FUNCTION_BLOCK FB_SetpointRamp
VAR_INPUT
    (* 斜坡运行许可。 *)
    bEnable : BOOL;
    (* 内部状态复位请求。 *)
    bReset : BOOL;
    (* 首次使能或复位后的连续起始值。 *)
    rInitialValue : LREAL;
    (* 需要平滑到达的目标值。 *)
    rTarget : LREAL;
    (* 正方向最大变化率，单位每秒。 *)
    rRateUpPer_s : LREAL;
    (* 负方向最大变化率绝对值，单位每秒。 *)
    rRateDownPer_s : LREAL;
    (* 实际调用周期，单位秒。 *)
    rCycleTime_s : LREAL;
    (* 判断到达目标的绝对容差。 *)
    rTolerance : LREAL;
END_VAR
VAR_OUTPUT
    (* 当前斜坡输出。 *)
    rOutput : LREAL;
    (* 仍在向目标变化时为TRUE。 *)
    bBusy : BOOL;
    (* 输出进入目标容差且不再需要变化时为TRUE。 *)
    bReached : BOOL;
    (* 周期、速率和输入均有效时为TRUE。 *)
    bValid : BOOL;
END_VAR
VAR
    (* 已用起始值建立连续输出。 *)
    bInitialized : BOOL;
    (* 所有可能影响输出的参数均有限且位于允许符号范围。 *)
    bInputsValid : BOOL;
    (* 非负到达容差。 *)
    rAbsoluteTolerance : LREAL;
END_VAR

bInputsValid := (rCycleTime_s > 0.0)
    AND (rRateUpPer_s >= 0.0)
    AND (rRateDownPer_s >= 0.0)
    AND (rTolerance >= 0.0)
    AND FC_IsFiniteLReal(rValue := rInitialValue)
    AND FC_IsFiniteLReal(rValue := rTarget)
    AND FC_IsFiniteLReal(rValue := rRateUpPer_s)
    AND FC_IsFiniteLReal(rValue := rRateDownPer_s)
    AND FC_IsFiniteLReal(rValue := rCycleTime_s)
    AND FC_IsFiniteLReal(rValue := rTolerance);

IF bReset OR NOT bEnable THEN
    IF bInputsValid THEN
        rOutput := rInitialValue;
    END_IF
    bInitialized := bEnable AND bInputsValid;
    bBusy := FALSE;
    bReached := FALSE;
    bValid := FALSE;
    IF NOT bEnable OR NOT bInputsValid THEN
        RETURN;
    END_IF
END_IF

bValid := bInputsValid;
IF NOT bValid THEN
    (* 参数无效时保持最后连续输出，不向设备发布跳变。 *)
    bBusy := FALSE;
    bReached := FALSE;
    RETURN;
END_IF

IF NOT bInitialized THEN
    rOutput := rInitialValue;
    bInitialized := TRUE;
END_IF

rOutput := FC_LimitRate(
    rCurrent := rOutput,
    rTarget := rTarget,
    rRateUpPer_s := rRateUpPer_s,
    rRateDownPer_s := rRateDownPer_s,
    rCycleTime_s := rCycleTime_s);
rAbsoluteTolerance := rTolerance;
bReached := ABS(rTarget - rOutput) <= rAbsoluteTolerance;
bBusy := NOT bReached;

END_FUNCTION_BLOCK

(* stored: Version 1.1.0.1
   POU FB_SetpointRamp: Id {B4000000-0000-4000-8000-000000000004} *)
